(* IEC 61131-3 sources: volt/packages/volt-lsp-iec/test-corpus/lenze-mid/Device/Plc Logic/Application/A71_LocalSources/CamControls/Window, 5 files *)

(* ---- fc_CamC_CC_Base.pou ---- *)
FUNCTION fc_CamC_CC_Base
VAR_INPUT
	i_xEnable				: BOOL;
	i_intStartCam			: INT;
	i_intStopCam			: INT;
	i_lrMachinePosition 	: LREAL;
END_VAR
VAR_OUTPUT
	o_xCamControl			: BOOL;
END_VAR
VAR
END_VAR

%LANGUAGE LD
%NETWORK
ASSIGN(BRANCH_SHORTCIRCUIT(FEED := i_xEnable, LE(EN := GE(EN := LT(EN := RAIL(), i_intStartCam, i_intStopCam).OUT, i_lrMachinePosition, i_intStartCam).OUT, i_lrMachinePosition, i_intStopCam).OUT, BRANCH_SHORTCIRCUIT(FEED := GT(EN := RAIL(), i_intStartCam, i_intStopCam).OUT, GE(EN := RAIL(), i_lrMachinePosition, i_intStartCam).OUT, LE(EN := RAIL(), i_lrMachinePosition, i_intStopCam).OUT)), Q => o_xCamControl);

END_FUNCTION

(* ---- fc_CamC_CC_UDT.pou ---- *)
FUNCTION fc_CamC_CC_UDT : bool
VAR_INPUT
	iEnable				: BOOL;
	iMachinePosition	: INT;

END_VAR

VAR
	tIndex:INT;
	B:INT;
	g:INT;
	E:INT;
	i:INT;
END_VAR
VAR_IN_OUT
	ioCamControl	: UDT_CamControl;
END_VAR

%LANGUAGE ST

ioCamControl.MachinePos_HMI:=iMachinePosition;
fc_CamC_CC_Base(
	i_xEnable:= 1,
	i_intStartCam:= ioCamControl.Start,
	i_intStopCam:=ioCamControl.Stop ,
	i_lrMachinePosition:=ioCamControl.MachinePos_HMI ,
	o_xCamControl=>fc_CamC_CC_UDT );

END_FUNCTION

(* ---- fc_CamC_LS_Base2.pou ---- *)
FUNCTION fc_CamC_LS_Base2 : bool
VAR_INPUT
	i_xEnable				: BOOL;
	i_intActualSpeed		: INT;
	i_intVLowSpeed			: INT;
	i_intVHighSpeed			: INT;
	i_intPosLowSpeedStart	: INT;
	i_intPosLowSpeedStop	: INT;
	i_intPosHighSpeedStart	: INT;
	i_intPosHighSpeedStop	: INT;
	i_lrActualMachPos	 	: LREAL;
END_VAR

VAR
	t_intPosLowSpeedStart	: INT;
	t_lrDY_Start			: LREAL;
	t_lrDX_Start			: LREAL;
	t_lrGain_Start			: LREAL;
	t_intToPosStart			: INT;
	t_intPosLowSpeedStop	: INT;
	t_lrDY_Stop				: LREAL;
	t_lrDX_Stop				: LREAL;
	t_lrGain_Stop			: LREAL;
	t_intToPosStop			: INT;
	xMemOutput				: BOOL;
	EdgeStart				: R_TRIG;
	EdgeStop				: R_TRIG;
	t_xStart				: BOOL;
	t_xStop					: BOOL;
	intMemStartPosition		: INT;
	intMemStopPosition		: INT;
END_VAR
VAR_IN_OUT
	OSP_START: BOOL;
	OSP_STOP: BOOL;
	FF_Started: BOOL;

END_VAR

%LANGUAGE ST
//START point: If HighSpeedPos>Lowspeed pos = zero is crossed, add 360
t_intPosLowSpeedStart := i_intPosLowSpeedStart;

IF i_intPosHighSpeedStart > t_intPosLowSpeedStart THEN
	t_intPosLowSpeedStart := (t_intPosLowSpeedStart + 360);
END_IF

//START point: Calculate angle (Gain) of interpolation
t_lrDY_Start := i_intPosHighSpeedStart - t_intPosLowSpeedStart;
t_lrDX_Start := i_intVHighSpeed - i_intVLowSpeed;
t_lrGain_Start := (t_lrDY_Start/t_lrDX_Start);

//START point: Calculate Startingpoint depending on actual speed
t_intToPosStart := LREAL_TO_INT(t_intPosLowSpeedStart + (t_lrGain_Start * (i_intActualSpeed - i_intVLowSpeed)));

IF t_intToPosStart >= 360 THEN
	t_intToPosStart := t_intToPosStart - 360;
ELSIF t_intToPosStart < 0 THEN
	t_intToPosStart := t_intToPosStart + 360;
END_IF

//STOP point: If HighSpeedPos>Lowspeed pos = zero is crossed, add 360
t_intPosLowSpeedStop := i_intPosLowSpeedStop;

IF i_intPosHighSpeedStop > t_intPosLowSpeedStop THEN
	t_intPosLowSpeedStop := (t_intPosLowSpeedStop + 360);
END_IF

//STOP point: Calculate angle (Gain) of interpolation
t_lrDY_Stop := i_intPosHighSpeedStop - t_intPosLowSpeedStop;
t_lrDX_Stop := i_intVHighSpeed - i_intVLowSpeed;
t_lrGain_Stop := (t_lrDY_Stop/t_lrDX_Stop);

//STOP point: Calculate stoppingpoint depending on actual speed
t_intToPosStop := LREAL_TO_INT(t_intPosLowSpeedStop + (t_lrGain_Stop * (i_intActualSpeed - i_intVLowSpeed)));

IF t_intToPosStop >= 360 THEN
	t_intToPosStop := t_intToPosStop - 360;
ELSIF t_intToPosStop < 0 THEN
	t_intToPosStop := t_intToPosStop + 360;
END_IF

//Actual position > START point -> set output
IF i_lrActualMachPos >= t_intToPosStart THEN
	t_xStart := TRUE;
ELSE
	t_xStart := FALSE;
END_IF

IF t_xStart <> OSP_START THEN
	FF_Started S= t_xStart;
	OSP_START:=t_xStart;
	IF FF_Started=TRUE THEN
		intMemStartPosition := t_intToPosStart;
	END_IF
END_IF

//Actual position > STOP point -> reset ouput
IF i_lrActualMachPos >= t_intToPosStop THEN
	t_xStop := TRUE;
ELSE
	t_xStop := FALSE;
END_IF

IF t_xStop <> OSP_STop THEN
	FF_Started R= t_xStop;
	OSP_STop:=t_xStop;
	IF FF_Started=FALSE THEN
		intMemStartPosition := t_intToPosStop;
	END_IF
END_IF

//Return 1 when in window
fc_CamC_LS_Base2 := FF_Started AND i_xEnable;

END_FUNCTION

(* ---- fc_CamC_LS_UDT.pou ---- *)
FUNCTION fc_CamC_LS_UDT : bool
VAR_INPUT
	iEnable			:  BOOL;
	iActualSpeed	:  INT;
	iActualPos		: INT;
	iRotflag 	: BOOL;
END_VAR
VAR
END_VAR

VAR_IN_OUT
	ioUDTCamControlLS	: UDT_CamControlLS;
END_VAR

%LANGUAGE LD
%NETWORK
MOVE(EN := RAIL(), iActualPos, OUT => ioUDTCamControlLS.MachinePos_HMI);
%NETWORK
ASSIGN(fc_CamC_LS_Base2(i_xEnable := RAIL(), i_intActualSpeed := iActualSpeed, i_intVLowSpeed := ioUDTCamControlLS.LowSpeed.SetSpeed, i_intVHighSpeed := ioUDTCamControlLS.HighSpeed.SetSpeed, i_intPosLowSpeedStart := ioUDTCamControlLS.LowSpeed.Start, i_intPosLowSpeedStop := ioUDTCamControlLS.LowSpeed.Stop, i_intPosHighSpeedStart := ioUDTCamControlLS.HighSpeed.Start, i_intPosHighSpeedStop := ioUDTCamControlLS.HighSpeed.Stop, i_lrActualMachPos := iActualPos, OSP_START := ioUDTCamControlLS.Calculation.OSStart, OSP_STOP := ioUDTCamControlLS.Calculation.OSStop, FF_Started := ioUDTCamControlLS.Calculation.FFStarted), Q => fc_CamC_LS_UDT);

END_FUNCTION

(* ---- fc_CamC_LS_Base.pou ---- *)
FUNCTION_BLOCK fc_CamC_LS_Base
VAR_INPUT
	i_xEnable				: BOOL;
	i_intActualSpeed		: INT;
	i_intVLowSpeed			: INT;
	i_intVHighSpeed			: INT;
	i_intPosLowSpeedStart	: INT;
	i_intPosLowSpeedStop	: INT;
	i_intPosHighSpeedStart	: INT;
	i_intPosHighSpeedStop	: INT;
	i_lrActualMachPos	 	: LREAL;
END_VAR
VAR_OUTPUT
	o_xCamControlLS			: BOOL;
END_VAR
VAR
	t_intPosLowSpeedStart	: INT;
	t_lrDY_Start			: LREAL;
	t_lrDX_Start			: LREAL;
	t_lrGain_Start			: LREAL;
	t_intToPosStart			: INT;
	t_intPosLowSpeedStop	: INT;
	t_lrDY_Stop				: LREAL;
	t_lrDX_Stop				: LREAL;
	t_lrGain_Stop			: LREAL;
	t_intToPosStop			: INT;
	xMemOutput				: BOOL;
	EdgeStart				: R_TRIG;
	EdgeStop				: R_TRIG;
	t_xStart				: BOOL;
	t_xStop					: BOOL;
	intMemStartPosition		: INT;
	intMemStopPosition		: INT;
END_VAR

%LANGUAGE ST
//START point: If HighSpeedPos>Lowspeed pos = zero is crossed, add 360
t_intPosLowSpeedStart := i_intPosLowSpeedStart;

IF i_intPosHighSpeedStart > t_intPosLowSpeedStart THEN
	t_intPosLowSpeedStart := (t_intPosLowSpeedStart + 360);
END_IF

//START point: Calculate angle (Gain) of interpolation
t_lrDY_Start := i_intPosHighSpeedStart - t_intPosLowSpeedStart;
t_lrDX_Start := i_intVHighSpeed - i_intVLowSpeed;
t_lrGain_Start := (t_lrDY_Start/t_lrDX_Start);

//START point: Calculate Startingpoint depending on actual speed
t_intToPosStart := LREAL_TO_INT(t_intPosLowSpeedStart + (t_lrGain_Start * (i_intActualSpeed - i_intVLowSpeed)));

IF t_intToPosStart >= 360 THEN
	t_intToPosStart := t_intToPosStart - 360;
ELSIF t_intToPosStart < 0 THEN
	t_intToPosStart := t_intToPosStart + 360;
END_IF

//STOP point: If HighSpeedPos>Lowspeed pos = zero is crossed, add 360
t_intPosLowSpeedStop := i_intPosLowSpeedStop;

IF i_intPosHighSpeedStop > t_intPosLowSpeedStop THEN
	t_intPosLowSpeedStop := (t_intPosLowSpeedStop + 360);
END_IF

//STOP point: Calculate angle (Gain) of interpolation
t_lrDY_Stop := i_intPosHighSpeedStop - t_intPosLowSpeedStop;
t_lrDX_Stop := i_intVHighSpeed - i_intVLowSpeed;
t_lrGain_Stop := (t_lrDY_Stop/t_lrDX_Stop);

//STOP point: Calculate stoppingpoint depending on actual speed
t_intToPosStop := LREAL_TO_INT(t_intPosLowSpeedStop + (t_lrGain_Stop * (i_intActualSpeed - i_intVLowSpeed)));

IF t_intToPosStop >= 360 THEN
	t_intToPosStop := t_intToPosStop - 360;
ELSIF t_intToPosStop < 0 THEN
	t_intToPosStop := t_intToPosStop + 360;
END_IF

//Actual position > START point -> set output
IF i_lrActualMachPos >= t_intToPosStart THEN
	t_xStart := TRUE;
ELSE
	t_xStart := FALSE;
END_IF

EdgeStart(CLK:= t_xStart);
xMemOutput S= EdgeStart.Q;

IF EdgeStart.Q = TRUE THEN
	intMemStartPosition := t_intToPosStart;
END_IF

//Actual position > STOP point -> reset ouput
IF i_lrActualMachPos >= t_intToPosStop THEN
	t_xStop := TRUE;
ELSE
	t_xStop := FALSE;
END_IF

EdgeStop(CLK:= t_xStop);
xMemOutput R= EdgeStop.Q;

IF EdgeStop.Q = TRUE THEN
	intMemStopPosition := t_intToPosStop;
END_IF

//Return 1 when in window
o_xCamControlLS := xMemOutput AND i_xEnable;

END_FUNCTION_BLOCK
